INTERFACE IStreamWriter

METHOD Add_BLOB : IStreamWriter
VAR_INPUT
    Value : ANY;
END_VAR
END_METHOD

METHOD Add_BOOL : IStreamWriter
VAR_INPUT
    Value : BOOL;
END_VAR
END_METHOD

METHOD Add_BYTE : IStreamWriter
VAR_INPUT
    Value : BYTE;
END_VAR
END_METHOD

METHOD Add_DINT : IStreamWriter
VAR_INPUT
    Value : DINT;
END_VAR
END_METHOD

METHOD Add_INT : IStreamWriter
VAR_INPUT
    Value : INT;
END_VAR
END_METHOD

METHOD Add_LINT : IStreamWriter
VAR_INPUT
    Value : LINT;
END_VAR
END_METHOD

METHOD Add_LREAL : IStreamWriter
VAR_INPUT
    Value : LREAL;
END_VAR
END_METHOD

METHOD Add_PVOID : IStreamWriter
VAR_INPUT
    Value : PVOID;
END_VAR
END_METHOD

METHOD Add_REAL : IStreamWriter
VAR_INPUT
    Value : REAL;
END_VAR
END_METHOD

METHOD Add_STRING : IStreamWriter
VAR_INPUT
    Value : STRING(255);
END_VAR
END_METHOD

METHOD Add_UDINT : IStreamWriter
VAR_INPUT
    Value : UDINT;
END_VAR
END_METHOD

METHOD Add_UINT : IStreamWriter
VAR_INPUT
    Value : UINT;
END_VAR
END_METHOD

METHOD Add_ULINT : IStreamWriter
VAR_INPUT
    Value : ULINT;
END_VAR
END_METHOD

METHOD Clear : IStreamWriter
END_METHOD

METHOD Seek: IStreamWriter
VAR_INPUT
    Position : UDINT;
END_VAR
END_METHOD

END_INTERFACE

(* stored: Version 1.1.0.1, ProductVersion 3.1.4024.3
   Itf IStreamWriter: Id {ade11aac-fe77-01bf-2404-d979d6533839}
   Folder Methods: Id {a77095f2-d0ea-0978-3d8c-52df480fa7c6}
   Method Add_BLOB: Id {b462fbbf-cc66-4f5b-9718-73f4255ea87b}
   Method Add_BOOL: Id {8cf5fe7f-aa12-004e-3325-fcee77aea2e1}
   Method Add_BYTE: Id {1d7ff7ed-48e4-01a6-29b6-deba0ee3a148}
   Method Add_DINT: Id {0a63b2b6-3995-06e0-1f6f-61ea68a48505}
   Method Add_INT: Id {b8297403-f002-0df9-1bfd-5cbf1d20c6b5}
   Method Add_LINT: Id {ceecd414-20fc-0ffc-297e-96b5b4c79cb7}
   Method Add_LREAL: Id {c0904514-c94e-035d-2758-34432039059e}
   Method Add_PVOID: Id {9d72da79-66b0-056e-0951-45e0c7dba648}
   Method Add_REAL: Id {c7ce2c7d-2413-0856-0f2a-b4514e497708}
   Method Add_STRING: Id {7241d1d3-a603-0390-3368-f88e5b224128}
   Method Add_UDINT: Id {b1a663c4-27ab-0810-24ef-9325bfd028e7}
   Method Add_UINT: Id {ff28e4a5-26e3-0df4-04d0-5fe2f1d49971}
   Method Add_ULINT: Id {4d97bc5e-9e02-0fee-2770-fbac7ae79b7d}
   Method Clear: Id {dd7f97e5-7e5a-00e5-30c5-73909163ad6b}
   Method Seek: Id {022de36b-fa7f-0b7c-1d93-83e7909f8ed3} *)
